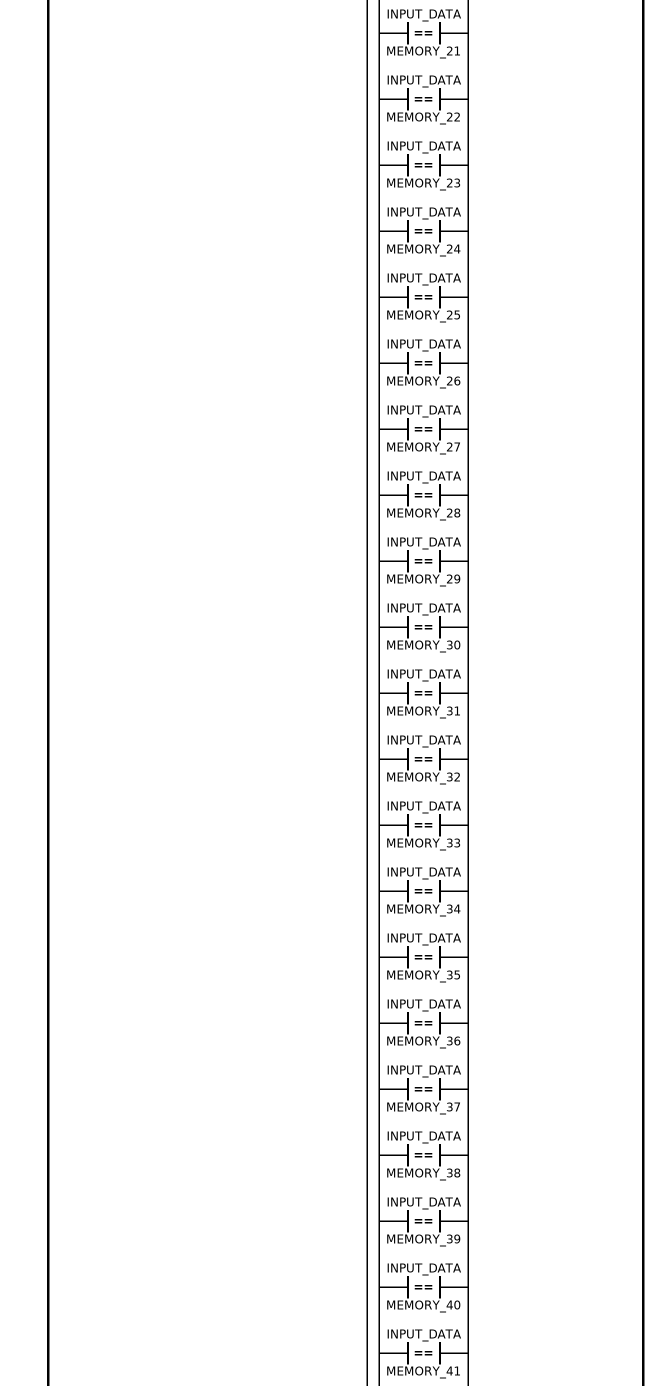
; [picture p120: FB RFID_SEQUENCE, rungs 8-8]

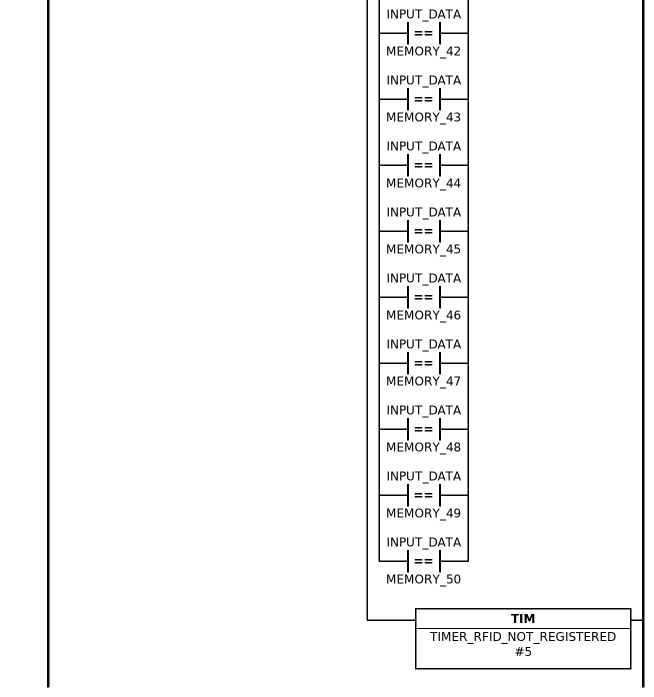
; rung 8
LD TIMER_RFID_READ_TIMEOUT
AND<>(305) INPUT_DATA #202D
AND<>(305) INPUT_DATA &0
OUT TR0
LD=(300) INPUT_DATA MEMORY_1
OR=(300) INPUT_DATA MEMORY_2
OR=(300) INPUT_DATA MEMORY_3
OR=(300) INPUT_DATA MEMORY_4
OR=(300) INPUT_DATA MEMORY_5
OR=(300) INPUT_DATA MEMORY_6
OR=(300) INPUT_DATA MEMORY_7
OR=(300) INPUT_DATA MEMORY_8
OR=(300) INPUT_DATA MEMORY_9
OR=(300) INPUT_DATA MEMORY_10
OR=(300) INPUT_DATA MEMORY_11
OR=(300) INPUT_DATA MEMORY_12
OR=(300) INPUT_DATA MEMORY_13
OR=(300) INPUT_DATA MEMORY_14
OR=(300) INPUT_DATA MEMORY_15
OR=(300) INPUT_DATA MEMORY_16
OR=(300) INPUT_DATA MEMORY_17
OR=(300) INPUT_DATA MEMORY_18
OR=(300) INPUT_DATA MEMORY_19
OR=(300) INPUT_DATA MEMORY_20
OR=(300) INPUT_DATA MEMORY_21
OR=(300) INPUT_DATA MEMORY_22
OR=(300) INPUT_DATA MEMORY_23
OR=(300) INPUT_DATA MEMORY_24
OR=(300) INPUT_DATA MEMORY_25
OR=(300) INPUT_DATA MEMORY_26
OR=(300) INPUT_DATA MEMORY_27
OR=(300) INPUT_DATA MEMORY_28
OR=(300) INPUT_DATA MEMORY_29
OR=(300) INPUT_DATA MEMORY_30
OR=(300) INPUT_DATA MEMORY_31
OR=(300) INPUT_DATA MEMORY_32
OR=(300) INPUT_DATA MEMORY_33
OR=(300) INPUT_DATA MEMORY_34
OR=(300) INPUT_DATA MEMORY_35
OR=(300) INPUT_DATA MEMORY_36
OR=(300) INPUT_DATA MEMORY_37
OR=(300) INPUT_DATA MEMORY_38
OR=(300) INPUT_DATA MEMORY_39
OR=(300) INPUT_DATA MEMORY_40
OR=(300) INPUT_DATA MEMORY_41
OR=(300) INPUT_DATA MEMORY_42
OR=(300) INPUT_DATA MEMORY_43
OR=(300) INPUT_DATA MEMORY_44
OR=(300) INPUT_DATA MEMORY_45
OR=(300) INPUT_DATA MEMORY_46
OR=(300) INPUT_DATA MEMORY_47
OR=(300) INPUT_DATA MEMORY_48
OR=(300) INPUT_DATA MEMORY_49
OR=(300) INPUT_DATA MEMORY_50
ANDLD
OUT RFID_CONFIRM_MATCH
LD TR0
TIM TIMER_RFID_NOT_REGISTERED #5

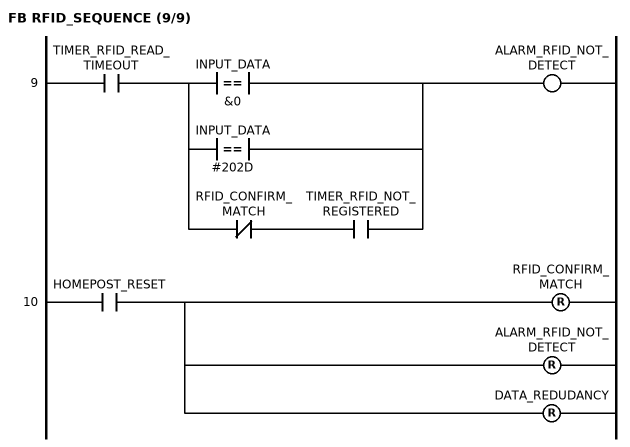
; rung 9
LD TIMER_RFID_READ_TIMEOUT
LD=(300) INPUT_DATA &0
OR=(300) INPUT_DATA #202D
LDNOT RFID_CONFIRM_MATCH
AND TIMER_RFID_NOT_REGISTERED
ORLD
ANDLD
OUT ALARM_RFID_NOT_DETECT
; rung 10
LD HOMEPOST_RESET
RSET RFID_CONFIRM_MATCH
RSET ALARM_RFID_NOT_DETECT
RSET DATA_REDUDANCY

## Function block ROTARY
VAR_INPUT
  PH_OUT : BOOL;
  PH_IN : BOOL;
  LS_STRAIGHT : BOOL;
  LS_TURN : BOOL;
  RS_PINLOCK_UP : BOOL;
  RS_PINLOCK_DOWN : BOOL;
  RS_STP_IN_UP : BOOL;
  RS_STP_IN_DOWN : BOOL;
  RS_STP_OUT_UP : BOOL;
  RS_STP_OUT_DOWN : BOOL;
  PH_OUT_CONVEYOR_BEFORE : BOOL;
  RS_STP_SIDE_CONV_DOWN : BOOL;
  PH_IN_CONVEYOR_AFTER : BOOL;
  PH_OUT_CONVEYOR_AFTER : BOOL;
  TURN_1 : BOOL;
  STRAIGHT_1 : BOOL;
  MOTOR_CONVEYOR_AFTER : BOOL;
  INTERLOCK_CONVEYOR_AFTER : BOOL;
  TON_PH_OUT_AFTER_OFF : BOOL;
  TRANSFER_FROM_CONV_BEFORE : BOOL;
  HOMEPOST_RESET : BOOL;
END_VAR
VAR_OUTPUT
  ROLL_IN_FWD : BOOL;
  ROLL_OUT_FWD : BOOL;
  MOTOR_ROT_FWD : BOOL;
  MOTOR_ROTARY_RVS : BOOL;
  PINLOCK_UP : BOOL;
  PINLOCK_DOWN : BOOL;
  STP_IN_UP : BOOL;
  STP_IN_DOWN : BOOL;
  STP_OUT_UP : BOOL;
  STP_OUT_DOWN : BOOL;
  DONE_STRAIGHT : BOOL;
  DONE_TURN : BOOL;
  TIMER_PH_OUT_AFTER_OFF : BOOL;
END_VAR
VAR
  MANUAL : BOOL;
  AUTO : BOOL;
  IR_CONFIRM_TURN : BOOL;
  CONFIRM_TRANSFER_TURN : BOOL;
  TIMEOUT_MROL_STP_IN : TIMER;
  TRANSFER_STRAIGHT_FROM_ROTARY : BOOL;
  TRANSFER_TURN_FROM_ROTARY : BOOL;
  MATERIAL_IN_ROTARY : BOOL;
  CONFIRM_TRANSFER_STRAIGHT : BOOL;
  MATERIAL_READY : BOOL;
  PINLOCK_DOWN_BEFORE_TURN : BOOL;
  ROTARY_TURN_FINISH : BOOL;
  PINLOCK_UP_AFTER_TURN : BOOL;
  ROTARY_STRAIGHT_AFTER_TURN : BOOL;
  PINLOCK_DOWN_AFTER_TURN : BOOL;
  PINLOCK_UP_AFTER_STRAIGHT : BOOL;
  DELAY_STP_IN_UP : TIMER;
END_VAR

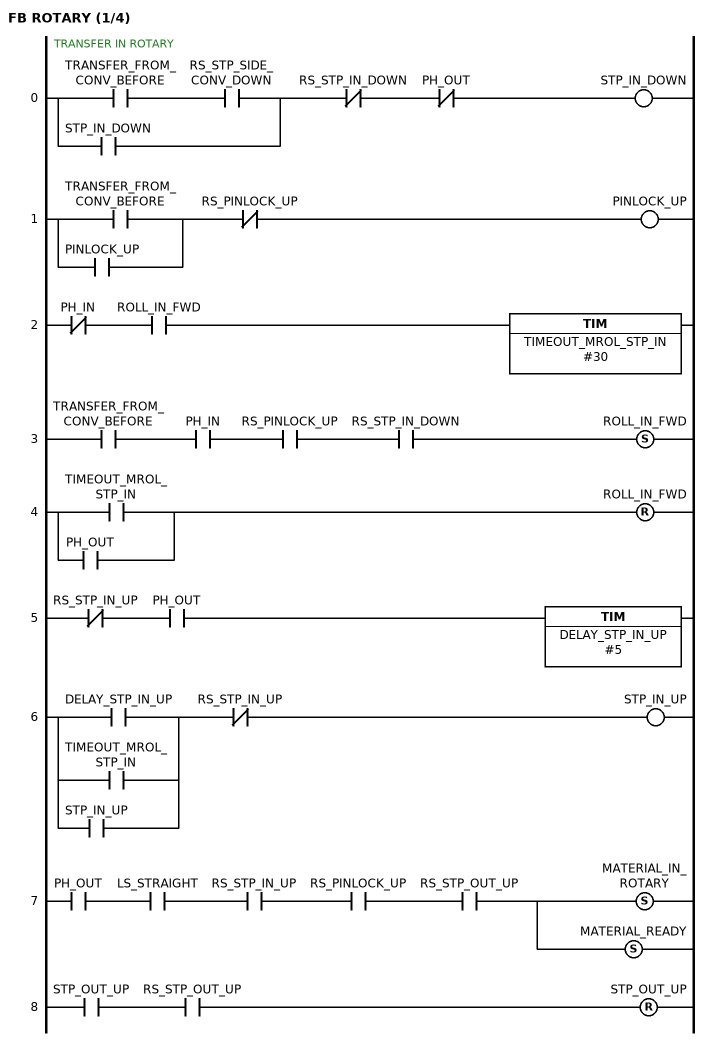
; rung 0: TRANSFER IN ROTARY
LD TRANSFER_FROM_CONV_BEFORE
AND RS_STP_SIDE_CONV_DOWN
OR STP_IN_DOWN
ANDNOT RS_STP_IN_DOWN
ANDNOT PH_OUT
OUT STP_IN_DOWN
; rung 1
LD TRANSFER_FROM_CONV_BEFORE
OR PINLOCK_UP
ANDNOT RS_PINLOCK_UP
OUT PINLOCK_UP
; rung 2
LDNOT PH_IN
AND ROLL_IN_FWD
TIM TIMEOUT_MROL_STP_IN #30
; rung 3
LD TRANSFER_FROM_CONV_BEFORE
AND PH_IN
AND RS_PINLOCK_UP
AND RS_STP_IN_DOWN
SET ROLL_IN_FWD
; rung 4
LD TIMEOUT_MROL_STP_IN
OR PH_OUT
RSET ROLL_IN_FWD
; rung 5
LDNOT RS_STP_IN_UP
AND PH_OUT
TIM DELAY_STP_IN_UP #5
; rung 6
LD DELAY_STP_IN_UP
OR TIMEOUT_MROL_STP_IN
OR STP_IN_UP
ANDNOT RS_STP_IN_UP
OUT STP_IN_UP
; rung 7
LD PH_OUT
AND LS_STRAIGHT
AND RS_STP_IN_UP
AND RS_PINLOCK_UP
AND RS_STP_OUT_UP
SET MATERIAL_IN_ROTARY
SET MATERIAL_READY
; rung 8
LD STP_OUT_UP
AND RS_STP_OUT_UP
RSET STP_OUT_UP

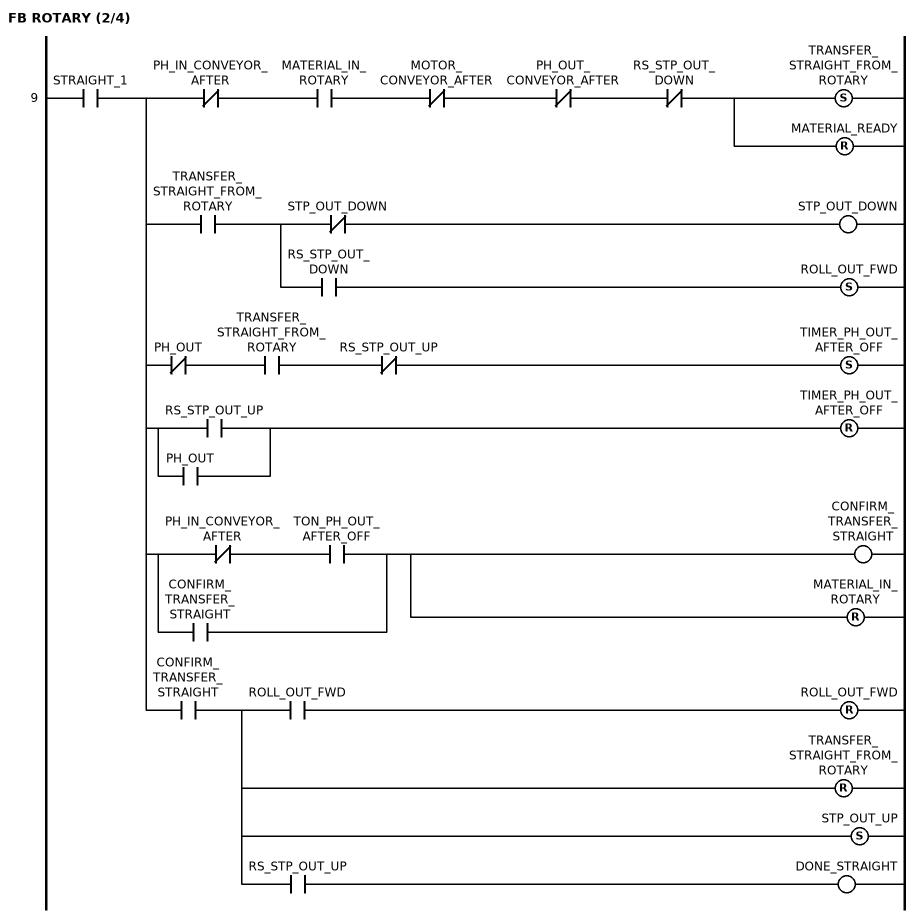
; rung 9
LD STRAIGHT_1
OUT TR0
ANDNOT PH_IN_CONVEYOR_AFTER
AND MATERIAL_IN_ROTARY
ANDNOT MOTOR_CONVEYOR_AFTER
ANDNOT PH_OUT_CONVEYOR_AFTER
ANDNOT RS_STP_OUT_DOWN
SET TRANSFER_STRAIGHT_FROM_ROTARY
RSET MATERIAL_READY
LD TR0
AND TRANSFER_STRAIGHT_FROM_ROTARY
OUT TR1
ANDNOT STP_OUT_DOWN
OUT STP_OUT_DOWN
LD TR1
AND RS_STP_OUT_DOWN
SET ROLL_OUT_FWD
LD TR0
ANDNOT PH_OUT
AND TRANSFER_STRAIGHT_FROM_ROTARY
ANDNOT RS_STP_OUT_UP
SET TIMER_PH_OUT_AFTER_OFF
LD TR0
LD RS_STP_OUT_UP
OR PH_OUT
ANDLD
RSET TIMER_PH_OUT_AFTER_OFF
LD TR0
LDNOT PH_IN_CONVEYOR_AFTER
AND TON_PH_OUT_AFTER_OFF
OR CONFIRM_TRANSFER_STRAIGHT
ANDLD
OUT CONFIRM_TRANSFER_STRAIGHT
RSET MATERIAL_IN_ROTARY
LD TR0
AND CONFIRM_TRANSFER_STRAIGHT
OUT TR2
AND ROLL_OUT_FWD
RSET ROLL_OUT_FWD
LD TR2
RSET TRANSFER_STRAIGHT_FROM_ROTARY
SET STP_OUT_UP
AND RS_STP_OUT_UP
OUT DONE_STRAIGHT

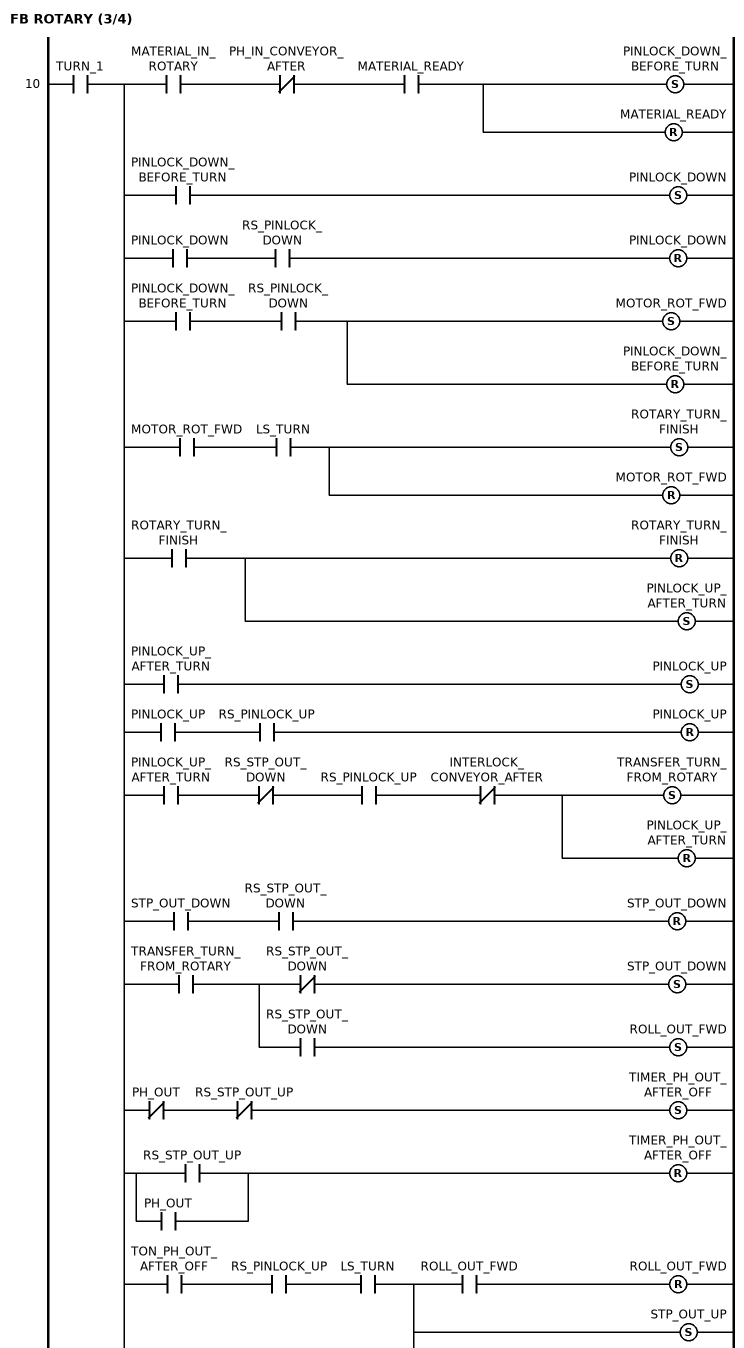

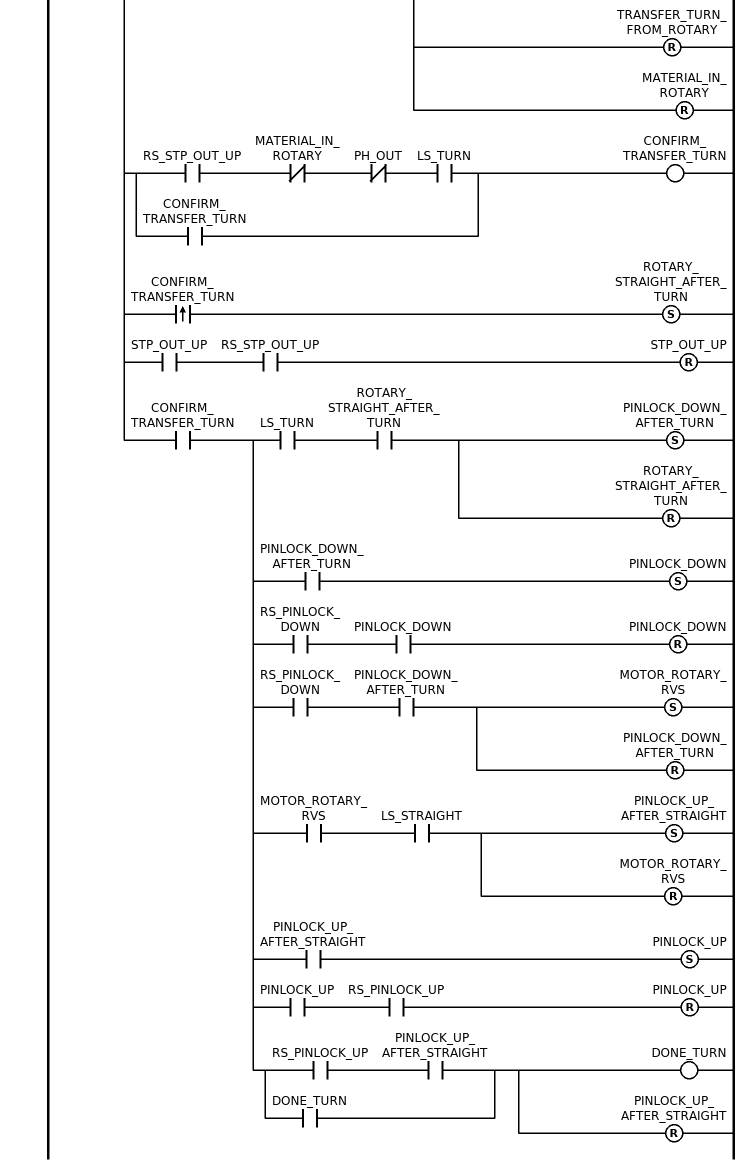
; rung 10
LD TURN_1
OUT TR0
AND MATERIAL_IN_ROTARY
ANDNOT PH_IN_CONVEYOR_AFTER
AND MATERIAL_READY
SET PINLOCK_DOWN_BEFORE_TURN
RSET MATERIAL_READY
LD TR0
AND PINLOCK_DOWN_BEFORE_TURN
SET PINLOCK_DOWN
LD TR0
AND PINLOCK_DOWN
AND RS_PINLOCK_DOWN
RSET PINLOCK_DOWN
LD TR0
AND PINLOCK_DOWN_BEFORE_TURN
AND RS_PINLOCK_DOWN
SET MOTOR_ROT_FWD
RSET PINLOCK_DOWN_BEFORE_TURN
LD TR0
AND MOTOR_ROT_FWD
AND LS_TURN
SET ROTARY_TURN_FINISH
RSET MOTOR_ROT_FWD
LD TR0
AND ROTARY_TURN_FINISH
RSET ROTARY_TURN_FINISH
SET PINLOCK_UP_AFTER_TURN
LD TR0
AND PINLOCK_UP_AFTER_TURN
SET PINLOCK_UP
LD TR0
AND PINLOCK_UP
AND RS_PINLOCK_UP
RSET PINLOCK_UP
LD TR0
AND PINLOCK_UP_AFTER_TURN
ANDNOT RS_STP_OUT_DOWN
AND RS_PINLOCK_UP
ANDNOT INTERLOCK_CONVEYOR_AFTER
SET TRANSFER_TURN_FROM_ROTARY
RSET PINLOCK_UP_AFTER_TURN
LD TR0
AND STP_OUT_DOWN
AND RS_STP_OUT_DOWN
RSET STP_OUT_DOWN
LD TR0
AND TRANSFER_TURN_FROM_ROTARY
OUT TR1
ANDNOT RS_STP_OUT_DOWN
SET STP_OUT_DOWN
LD TR1
AND RS_STP_OUT_DOWN
SET ROLL_OUT_FWD
LD TR0
ANDNOT PH_OUT
ANDNOT RS_STP_OUT_UP
SET TIMER_PH_OUT_AFTER_OFF
LD TR0
LD RS_STP_OUT_UP
OR PH_OUT
ANDLD
RSET TIMER_PH_OUT_AFTER_OFF
LD TR0
AND TON_PH_OUT_AFTER_OFF
AND RS_PINLOCK_UP
AND LS_TURN
OUT TR2
AND ROLL_OUT_FWD
RSET ROLL_OUT_FWD
LD TR2
SET STP_OUT_UP
RSET TRANSFER_TURN_FROM_ROTARY
RSET MATERIAL_IN_ROTARY
LD TR0
LD RS_STP_OUT_UP
ANDNOT MATERIAL_IN_ROTARY
ANDNOT PH_OUT
AND LS_TURN
OR CONFIRM_TRANSFER_TURN
ANDLD
OUT CONFIRM_TRANSFER_TURN
LD TR0
@AND CONFIRM_TRANSFER_TURN
SET ROTARY_STRAIGHT_AFTER_TURN
LD TR0
AND STP_OUT_UP
AND RS_STP_OUT_UP
RSET STP_OUT_UP
LD TR0
AND CONFIRM_TRANSFER_TURN
OUT TR3
AND LS_TURN
AND ROTARY_STRAIGHT_AFTER_TURN
SET PINLOCK_DOWN_AFTER_TURN
RSET ROTARY_STRAIGHT_AFTER_TURN
LD TR3
AND PINLOCK_DOWN_AFTER_TURN
SET PINLOCK_DOWN
LD TR3
AND RS_PINLOCK_DOWN
AND PINLOCK_DOWN
RSET PINLOCK_DOWN
LD TR3
AND RS_PINLOCK_DOWN
AND PINLOCK_DOWN_AFTER_TURN
SET MOTOR_ROTARY_RVS
RSET PINLOCK_DOWN_AFTER_TURN
LD TR3
AND MOTOR_ROTARY_RVS
AND LS_STRAIGHT
SET PINLOCK_UP_AFTER_STRAIGHT
RSET MOTOR_ROTARY_RVS
LD TR3
AND PINLOCK_UP_AFTER_STRAIGHT
SET PINLOCK_UP
LD TR3
AND PINLOCK_UP
AND RS_PINLOCK_UP
RSET PINLOCK_UP
LD TR3
LD RS_PINLOCK_UP
AND PINLOCK_UP_AFTER_STRAIGHT
OR DONE_TURN
ANDLD
OUT DONE_TURN
RSET PINLOCK_UP_AFTER_STRAIGHT

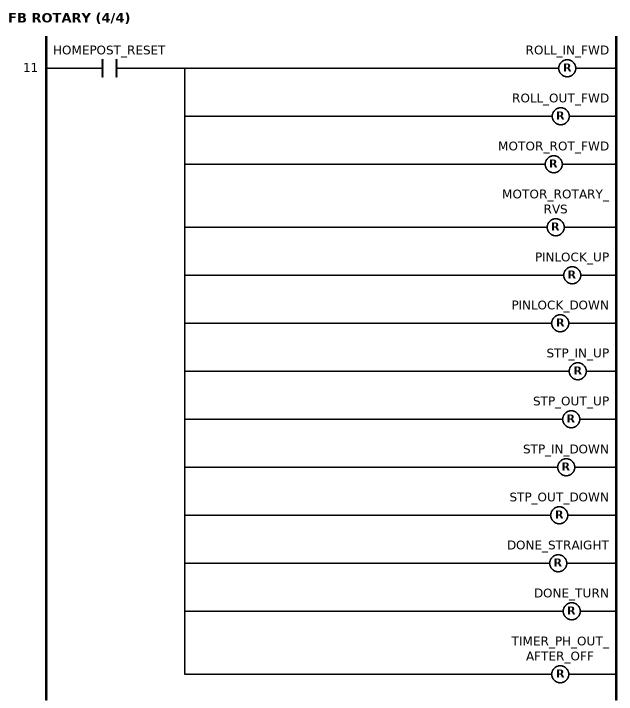
; rung 11
LD HOMEPOST_RESET
RSET ROLL_IN_FWD
RSET ROLL_OUT_FWD
RSET MOTOR_ROT_FWD
RSET MOTOR_ROTARY_RVS
RSET PINLOCK_UP
RSET PINLOCK_DOWN
RSET STP_IN_UP
RSET STP_OUT_UP
RSET STP_IN_DOWN
RSET STP_OUT_DOWN
RSET DONE_STRAIGHT
RSET DONE_TURN
RSET TIMER_PH_OUT_AFTER_OFF